Staubli VAL3: iCryoLongIn.pgx

public program iCryoLongIn(num& nNum[] (dimensions=1))
begin
  nNum=dioGet(iCryoLongIn)
end
